// TIA Portal project "Forno" (V14)

(* hardware
DEVICE "S7-1200 station_1"  S7-1200 Station
   slot 0: "Rack_0"  Rack  V1.0
   slot 1: "PLC_1"  CPU 1214C DC/DC/DC  6ES7 214-1AG31-0XB0  V3.0
*)

// ===== PLC "PLC_1"  CPU 1214C DC/DC/DC =====

VAR_GLOBAL   // PLC tag table "Default tag table"
   "Pressostato_alta" AT %M0.0 : Bool;
   "Pressostato_baixa" AT %M0.1 : Bool;
   "Fluxo_exaust" AT %M0.2 : Bool;
   "Fluxo_forc" AT %M0.3 : Bool;
   "porta_closed" AT %M0.4 : Bool;
   "porta_opened" AT %M0.5 : Bool;
   "chama_piloto" AT %M0.6 : Bool;
   "chama_pricipal" AT %M0.7 : Bool;
   "Relay_chama_ok" AT %M1.0 : Bool;
   "Vent_exaust" AT %Q0.0 : Bool;
   "Vent_forc" AT %Q0.1 : Bool;
   "open_porta" AT %Q0.2 : Bool;
   "close_porta" AT %Q0.3 : Bool;
   "Valv_controle" AT %Q0.4 : Bool;
   "Bloqueio" AT %Q0.5 : Bool;
END_VAR

ORGANIZATION_BLOCK "Main"   // OB1, LAD, ProgramCycle
TITLE = "Main Program Sweep (Cycle)"
{ S7_Optimized_Access := 'TRUE' }
VERSION : 0.1
BEGIN
END_ORGANIZATION_BLOCK